// Mitsubishi GX Works2 project: Joystickövn   PLC: Q03UDE

// global labels: Global1
VAR_GLOBAL
  Start AT X0 : BOOL;
  J2_0 AT X2 : BOOL;
  Steg_1 : BOOL;
  J2_90 AT X3 : BOOL;
  Steg_2 : BOOL;
  TimerMinne2 : BOOL;
  TimerMinne1 : BOOL;
  J2_270 AT X5 : BOOL;
  Steg_3 : BOOL;
  Framme : BOOL;
  J2_180 AT X4 : BOOL;
  TimerMinne3 : BOOL;
  J1_180 AT X8 : BOOL;
  Steg_4 : BOOL;
  J1_0 AT X6 : BOOL;
  Steg_5 : BOOL;
  TimerMinne4 : BOOL;
  Stopp AT X1 : BOOL;
  J1_270 AT X9 : BOOL;
  Steg_6 : BOOL;
  J1_90 AT X7 : BOOL;
  Hemma : BOOL;
  MotorFram AT Y0 : BOOL;
  Lo AT Y2 : BOOL;
  Grön AT Y5 : BOOL;
  MotorBack AT Y1 : BOOL;
  Vit AT Y6 : BOOL;
  Röd AT Y7 : BOOL;
  Md AT Y3 : BOOL;
  Hi AT Y4 : BOOL;
  Cyl1_UT AT Y8 : BOOL;
  Cyl2_UT AT Y10 : BOOL;
  Cyl1_IN AT Y9 : BOOL;
  Cyl2_IN AT Y11 : BOOL;
  Cyl1_INNE AT X10 : BOOL;
  Cyl2_INNE AT X11 : BOOL;
END_VAR

PROGRAM Sekvens
VAR
  Kör : BOOL;
  Timer_01 : TON;
  Timer_02 : TON;
  Timer_03 : TON;
  Timer_04 : TON;
END_VAR
(* structured ladder/FBD written out as ST: instructions are called as NAME(EN, inputs, outputs); _pN, _eN, _tN stand for wires *)
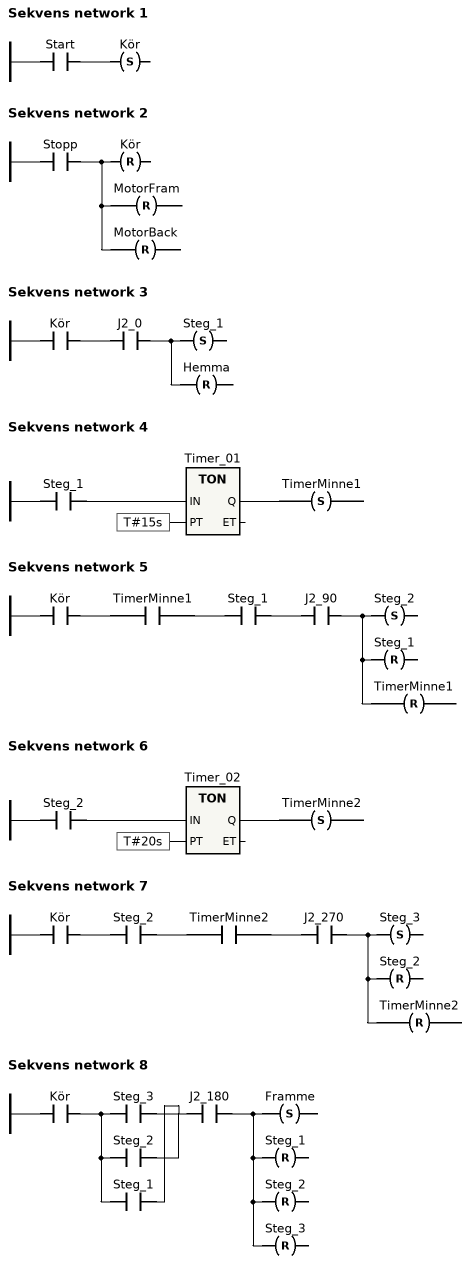
(* network 1 *)
SET(Start, Kör);
(* network 2 *)
RST(Stopp, Kör);
RST(Stopp, MotorFram);
RST(Stopp, MotorBack);
(* network 3 *)
_p1 := Kör AND J2_0;
SET(_p1, Steg_1);
RST(_p1, Hemma);
(* network 4 *)
Timer_01(IN := Steg_1, PT := T#15s);
SET(Timer_01.Q, TimerMinne1);
(* network 5 *)
_p1 := Kör AND TimerMinne1 AND Steg_1 AND J2_90;
SET(_p1, Steg_2);
RST(_p1, Steg_1);
RST(_p1, TimerMinne1);
(* network 6 *)
Timer_02(IN := Steg_2, PT := T#20s);
SET(Timer_02.Q, TimerMinne2);
(* network 7 *)
_p1 := Kör AND Steg_2 AND TimerMinne2 AND J2_270;
SET(_p1, Steg_3);
RST(_p1, Steg_2);
RST(_p1, TimerMinne2);
(* network 8 *)
_p1 := ((Kör AND Steg_3) OR (Kör AND Steg_2) OR (Kör AND Steg_1)) AND J2_180;
SET(_p1, Framme);
RST(_p1, Steg_1);
RST(_p1, Steg_2);
RST(_p1, Steg_3);
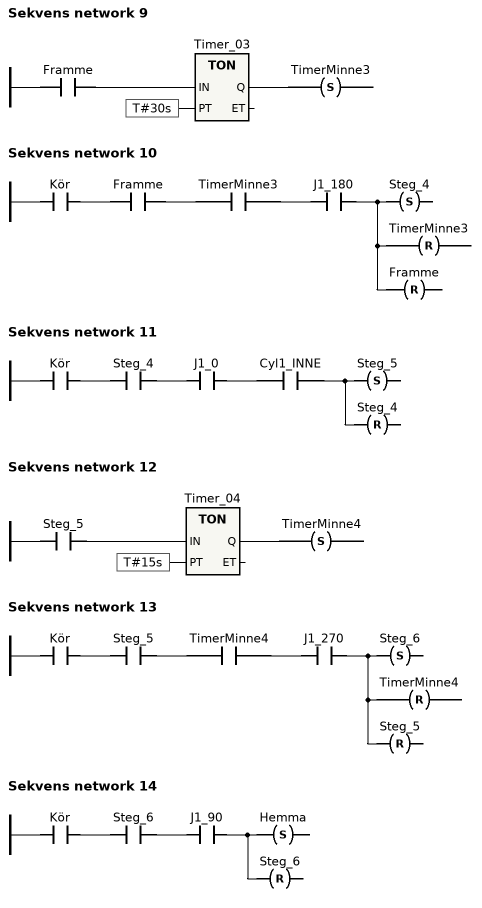
(* network 9 *)
Timer_03(IN := Framme, PT := T#30s);
SET(Timer_03.Q, TimerMinne3);
(* network 10 *)
_p1 := Kör AND Framme AND TimerMinne3 AND J1_180;
SET(_p1, Steg_4);
RST(_p1, TimerMinne3);
RST(_p1, Framme);
(* network 11 *)
_p1 := Kör AND Steg_4 AND J1_0 AND Cyl1_INNE;
SET(_p1, Steg_5);
RST(_p1, Steg_4);
(* network 12 *)
Timer_04(IN := Steg_5, PT := T#15s);
SET(Timer_04.Q, TimerMinne4);
(* network 13 *)
_p1 := Kör AND Steg_5 AND TimerMinne4 AND J1_270;
SET(_p1, Steg_6);
RST(_p1, TimerMinne4);
RST(_p1, Steg_5);
(* network 14 *)
_p1 := Kör AND Steg_6 AND J1_90;
SET(_p1, Hemma);
RST(_p1, Steg_6);
END_PROGRAM

PROGRAM Aktivering
(* structured ladder/FBD written out as ST: instructions are called as NAME(EN, inputs, outputs); _pN, _eN, _tN stand for wires *)
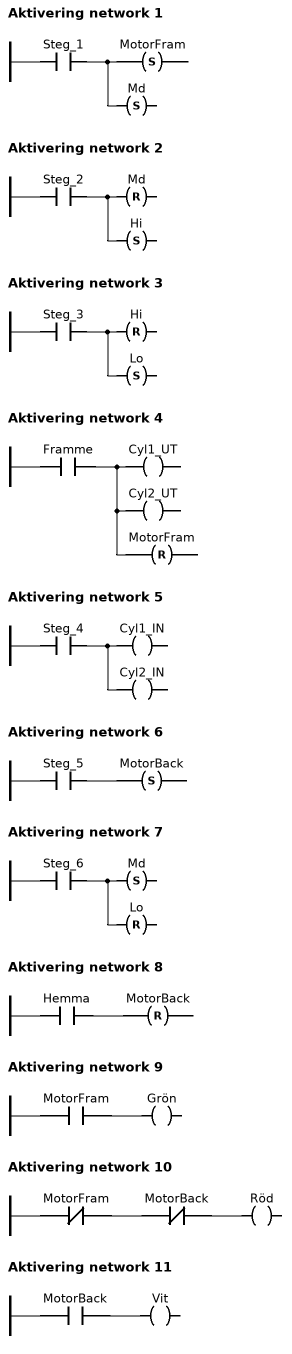
(* network 1 *)
SET(Steg_1, MotorFram);
SET(Steg_1, Md);
(* network 2 *)
RST(Steg_2, Md);
SET(Steg_2, Hi);
(* network 3 *)
RST(Steg_3, Hi);
SET(Steg_3, Lo);
(* network 4 *)
Cyl1_UT := Framme;
Cyl2_UT := Framme;
RST(Framme, MotorFram);
(* network 5 *)
Cyl1_IN := Steg_4;
Cyl2_IN := Steg_4;
(* network 6 *)
SET(Steg_5, MotorBack);
(* network 7 *)
SET(Steg_6, Md);
RST(Steg_6, Lo);
(* network 8 *)
RST(Hemma, MotorBack);
(* network 9 *)
Grön := MotorFram;
(* network 10 *)
Röd := NOT MotorFram AND NOT MotorBack;
(* network 11 *)
Vit := MotorBack;
END_PROGRAM
